(* PLC project BlogProject.project, CODESYS CODESYS V3.5 SP14 Patch 3 *)
(* stored: creationDateTime 2021-10-07T21:07:30.7532792, modificationDateTime 2021-10-07T20:40:20.1109198 *)

FUNCTION_BLOCK mcStartSystem IMPLEMENTS itfAction
  VAR_OUTPUT
    SystemStart : BOOL;
  END_VAR

            
          

METHOD getAction : BOOL
                  SystemStart:=TRUE;
StartCommand:=FALSE;
                
END_METHOD
END_FUNCTION_BLOCK
